# EPICS autosave request: iocBoot/sioc-li20-im03/sioc-li20-im03.req
file "facet2.req" AREA=LI20,POS=3255
